Staubli VAL3: Poche.pgx

program Poche(pointRx x_pStartPoint, num x_nDiametreTool, num x_nPasseAxiale, num x_nPasseRadiale, num x_nDimX, num x_nDimY, num x_nDimZ)
  local num l_nIndex
  local pointRx l_pPoint[5]
  local num l_nIndex2
  local num l_nN
  local num l_nLongueurCote
  local num l_nIndex3
  local num l_nM
  local num l_nProfondeur
begin
  logMsg("Beginning...")

  l_nProfondeur = x_nDimZ

  l_nN = roundDown((x_nDimX-x_nDiametreTool-x_nPasseRadiale)/(2*x_nPasseRadiale)+1)
  l_nM = roundDown(l_nProfondeur/(x_nPasseAxiale))

  for l_nIndex3 = 1 to l_nM
    logMsg("New passe...")
    if l_nIndex3 == l_nM
      l_pPoint[0] = appro(x_pStartPoint,{x_nDiametreTool/2,x_nDiametreTool/2,l_nProfondeur,0,0,0})
    else
      l_pPoint[0] = appro(x_pStartPoint,{x_nDiametreTool/2,x_nDiametreTool/2,l_nIndex3 * x_nPasseAxiale,0,0,0})
    endIf
    movej(appro(l_pPoint[0],trAppro), tBroche, mRapide100On)

    movel(l_pPoint[0], tBroche, mUsinage20Off)

    //------------------------------------- Forme centrale ------------------------------------------------
    for l_nIndex = 0 to l_nN - 1
      l_pPoint[1] = compose(l_pPoint[0], fPiece, {l_nIndex*2*x_nPasseRadiale,0,0,0,0,0})
      l_pPoint[2] = compose(l_pPoint[1], fPiece, {0,x_nDimY - x_nDiametreTool,0,0,0,0})
      l_pPoint[3] = compose(l_pPoint[2], fPiece, {x_nPasseRadiale,0,0,0,0,0})
      l_pPoint[4] = compose(l_pPoint[3], fPiece, {0,-(x_nDimY - x_nDiametreTool),0,0,0,0})

      for l_nIndex2 = 1 to 4
        movel(l_pPoint[l_nIndex2], tBroche, mUsinage20Off)
      endFor
    endFor
    logMsg("Last 'U'")
    l_pPoint[1] = compose(l_pPoint[0], fPiece, {(x_nDimX - x_nDiametreTool) -  x_nPasseRadiale,0,0,0,0,0})
    l_pPoint[2] = compose(l_pPoint[1], fPiece, {0,x_nDimY - x_nDiametreTool,0,0,0,0})
    l_pPoint[3] = compose(l_pPoint[2], fPiece, {x_nPasseRadiale,0,0,0,0,0})
    l_pPoint[4] = compose(l_pPoint[3], fPiece, {0,-(x_nDimY - x_nDiametreTool),0,0,0,0})

    for l_nIndex2 = 1 to 4
      movel(l_pPoint[l_nIndex2], tBroche, mUsinage20Off)
    endFor

    //------------------------------------- Forme contours ------------------------------------------------

    movel(l_pPoint[0], tBroche, mUsinage20Off)
    movel(appro(l_pPoint[0],trAppro), tBroche, mUsinage20Off)

    l_pPoint[1] = compose(l_pPoint[0], fPiece, {0,x_nDimY - x_nDiametreTool,0,0,0,0})
    l_pPoint[2] = compose(l_pPoint[1], fPiece, {x_nDimX - x_nDiametreTool,0,0,0,0,0})

    movej(appro(l_pPoint[1], trAppro), tBroche, mRapide100On)
    movel(l_pPoint[1], tBroche, mUsinage20Off)
    movel(l_pPoint[2], tBroche, mUsinage20Off)
    movel(appro(l_pPoint[2], trAppro), tBroche, mUsinage20Off)
  endFor
  movej(appro(l_pPoint[0],trAppro), tBroche, mRapide100On)
  logMsg("Program ended.")
end
